TYPE (* IEC61131-3, Table 14#5 *)
  (* Standard: 1131-3 *)
  (* Version 0.0, 1/8/2024, Cheyan, Schneider Electric, Template *)
  PACKAGE Main;
  {SET_ATTRIBUTE(nxtDataType, /vixPIdCcZLsYuYBrz+XyN166j18T5K4HgXF1dcTzTZHQJ1wIsOj+9aXLW6JvpI5liIDCK+YB6XbIe7VaGVjE0bwToVoS8iyEAyKPLQdQVMhZA8RLgefo7Yx7v7UbzEoNi1L3qeHb/EumZ+i8RhQUi+lIU4Z/rct1mfeorKNTf4ZIwa2bBiI8A==)}
  DPC : STRUCT
    stVal : stVal;
    q : Quality;
    t : TimeStamp;
    CtlModel : CtlModels;
  END_STRUCT;
END_TYPE
